Staubli VAL3: ClientSend.pgx

public program ClientSend(string x_sMess)
begin
  sClient=x_sMess
end
